(*
  Managing a production on a DigiRound machine.
*)
FUNCTION_BLOCK FB_ProdManager_DMAX EXTENDS FB_BasePrint IMPLEMENTS I_PrintStatusClient, I_ProdManager
VAR
 //references
  _pPU                : POINTER TO FB_PU;               (*PU reference*)
  _pAdsPU             : POINTER TO ST_ADS_PU;
  
  //settings
  _defaultPrintData   : ST_PRINT_SETTING;               (*default PDI data if no CT present*)
  _isVarData          : BOOL; 

  //status
  bPmActive           : BOOL;                           (*a production is active*)
  rfTrig_PmActive     : RF_TRIG;
  lastCreatedCT       : I_CT;                           (*last created container*)

  (*lists*)
  (*--list implementations*)
  prodList            : FB_ListPointerDyn;              (*list fb [pointer to I_CT] - current production elements*)
  _prodMem            : ARRAY[1..lNUM_LIST_SIZE] OF PVOID;   (*list memory for prodList*)
  (*--job trace list*)
  _currJobId          : STRING;                         (*id of current started job*)

  (*internals*)
  _pEcSrc : POINTER TO T_ErrSrc;                                    (*error source definition*)

END_VAR
VAR CONSTANT
  lNUM_LIST_SIZE        : DINT := iCPr_MAX_CONTAINER;   (*number of max. list elements*)
  // other logs
  aC_Dbg_NotReject      : STRING := 'could not rejectNext CT';
  aC_Dbg_InvPtrCT       : STRING := 'invalid pO_ContainerHead';
  aC_Dbg_InvPtrJob      : STRING := 'invalid Job pointer';
  aC_Ddb_GetNext        : STRING := 'getNext from: ';  
END_VAR

IF NOT bInitialized THEN RETURN; END_IF  // ignore

rfTrig_PmActive(CLK:=bPmActive);

(*
  Job was stopped. 
  :return: TRUE if some elements were aborted in machine.
*)
METHOD PRIVATE abortJob : BOOL
VAR
END_VAR
// a job stopped.

// NOTE: not implemented
END_METHOD

PROPERTY bReady : BOOL
GET
bReady := bPmActive;
END_GET
END_PROPERTY

PROPERTY bStarted : BOOL
GET
bStarted := rfTrig_PmActive.RT;
END_GET
END_PROPERTY

PROPERTY bStopped : BOOL
GET
bStopped := rfTrig_PmActive.FT;
END_GET
END_PROPERTY

(*
Create/Build a new container (CT) with next page to be printed.
*)
METHOD CT_Create : BOOL
VAR_INPUT
  sCT            : I_CT;                  // container to produce
END_VAR
VAR 
  _created       : BOOL := FALSE;
  sPage          : ST_PrintPageDef;
END_VAR
// prepare & checks
lastCreatedCT := 0;                      // invalidate last created
IF NOT bInitialized THEN RETURN; END_IF
IF sCT = 0 THEN LogError(aC_Dbg_InvPtrCT); RETURN; END_IF

(* getNext CT *)
IF getNext(sCT := sCT) THEN
  
  // define printer output
  sPage := sCT.sPageDef;
  IF    sPage.lType = EN_PrintPageType.maintenance THEN // - maintenance
    sCT.pCT^.lPrOutput := EN_PrinterOutput.trash;     // -> eject trash
  ELSIF sPage.lType = EN_PrintPageType.production OR   // - production
        sPage.lSrc = EN_PrintPageSrc.overprod OR       // - over-production
        sPage.lType = EN_PrintPageType.separator THEN  // - separator 
    sCT.pCT^.lPrOutput := EN_PrinterOutput.prod;      // -> production output
  ELSE                                                // - rest
    sCT.pCT^.lPrOutput := EN_PrinterOutput.trash;     // -> eject trash
  END_IF

  lastCreatedCT := sCT;                // successfully produced a CT, store last created CT (necessary for async access within this cycle)
  sCT.pCT^.bCreated := TRUE;
  _created := TRUE;
ELSE
  sCT.setError(EC_Print.ecPMInvGetNext, Src:=_pEcSrc^);   // getNext error
END_IF

(* logging *)
LogLvl(Lvl:=E_LogSeverity.Debug, Msg:=CONCAT('create CT: ', sCT.print(0)));

(*return value*)
CT_Create := _created;
END_METHOD

METHOD CT_Finish : BOOL
VAR_INPUT
  sCT            : I_CT;               // container to produce
  bSuccess       : BOOL;               // printed OK?
END_VAR
VAR
  bErr           : BOOL;
END_VAR
(* checks *)
IF NOT bInitialized THEN RETURN; END_IF                             // exit if no production is active
IF sCT = 0 THEN LogError(aC_Dbg_InvPtrCT); RETURN; END_IF  // log invalid pointer 

// remove from production list
IF NOT prodList.RemoveIndex(prodList.FindIndex(sCT.instance)) THEN
  LogError('CT_Finish: could not find CT in prodList'); 
END_IF

// tag machine errors on CT
IF sCT.pCT^.bValid AND NOT bSuccess THEN  
    sCT.setError(EC_Print.ecPMCTMachineErr, Src:=_pEcSrc^);            // tag CT with: error from machine 
END_IF

// report page done to PU
IF NOT sCT.pCT^.bReported AND sCT.pJob <> 0 THEN
  IF _pPU^.endPage(sCT:=sCT, bSuccess:=bSuccess) THEN
    ;
  ELSE
    sCT.setError(EC_Print.ecPMInvSet, Src:=_pEcSrc^);
  END_IF
END_IF

(* logging *)
IF bSuccess THEN
  LogLvl(Lvl:=E_LogSeverity.Detail, Msg:=CONCAT('successCT: ', sCT.print(0)));
ELSE
  LogLvl(Lvl:=E_LogSeverity.Detail, Msg:=CONCAT('eject  CT: ', sCT.print(0)));  
END_IF

(* return value *)
CT_Finish := TRUE;
END_METHOD

(*
  Finalize/Produce a CT. Now we shouldhave all necessary information for configuring the CT.
*)
METHOD CT_Produce : BOOL
VAR_INPUT
  sCT                 : I_CT;               // container to produce
END_VAR
VAR
  _produced           : BOOL := FALSE;
  sPage               : ST_PrintPageDef;
  bPresent            : BOOL;
END_VAR
(* parameter checks *)
IF NOT bInitialized THEN RETURN; END_IF
IF sCT = 0 THEN LogError(aC_Dbg_InvPtrCT); RETURN; END_IF

sCT.pCT^.bValid           := TRUE;                (* we have all data - CT is valid configured*)

// reject page if no container present or overproduction
sPage := sCT.sPageDef;
bPresent := sCT.pCT^.bProductPresent;
IF NOT bPresent AND sPage.lSrc <> EN_PrintPageSrc.overprod  THEN
  (*   add it to rejected queue (high prio reproduction), we will try to produce this CT in next cycle*)
  IF NOT _pPU^.rejPage(sCT:=sCT) THEN
    LogLvl(Lvl:=E_LogSeverity.Info, aC_Dbg_NotReject);
  END_IF
END_IF

(* logging *)
IF bPresent THEN LogLvl(Lvl:=E_LogSeverity.Detail,  Msg:=CONCAT('produceCT: ', sCT.print(0)));
            ELSE LogLvl(Lvl:=E_LogSeverity.Debug,   Msg:=CONCAT('produceCT: ', sCT.print(0))); END_IF

(* return value*)
CT_Produce := _produced;
END_METHOD

PROPERTY defaultPrData : ST_PRINT_SETTING
GET
defaultPrData := _defaultPrintData;
END_GET
END_PROPERTY

METHOD PRIVATE dynAddPage : BOOL
VAR_INPUT
  lType     : EN_PrintPageType; 
  lPageNr   : UDINT;
END_VAR
IF _pPU = 0 THEN F_Report_Error(ErrType:=EN_REPORT_ERROR_TYPE.Report_Error_0Pointer); RETURN; END_IF
IF lType <> EN_PrintPageType.maintenance THEN
  LogError('dynAddPage: only supports maintenance pages'); 
END_IF

_pPU^.addPage(lMaintPageNr:=lPageNr);
END_METHOD

(*
  get next page to be printed.
  :return:    TRUE if success.
*)
METHOD PRIVATE getNext : BOOL               (*get next image to be printed*)
VAR_INPUT
  sCT               : I_CT;                 (*container handle*)
END_VAR
VAR
  bErr              : BOOL;
  lRemainingPages   : UDINT;
END_VAR
VAR_INST
  rTrig_PreStop     : R_TRIG;
END_VAR
IF NOT bInitialized THEN RETURN; END_IF                    (* Exit if no production is active*)

// ask pu for a next page
bErr := NOT _pPU^.getPage(sCT:=sCT, lPagesLeft=>lRemainingPages);

// add to producing list
IF NOT prodList.AddItem(Item := sCT.instance) THEN 
  LogError('getNext: could not add CT to prodList');
  bErr := TRUE;
END_IF

getNext := NOT bErr;
END_METHOD

METHOD init : BOOL
VAR_INPUT
  pPU     : POINTER TO FB_PU;
  pAdsPU  : POINTER TO ST_ADS_PU;
  // machine specific
END_VAR
// parameter checks
IF pPU = 0 OR pAdsPU = 0 THEN
  F_Report_Error(ErrType:=EN_REPORT_ERROR_TYPE.Report_Error_0Pointer);
  RETURN;
END_IF

// register external references
_pPU := pPU;
_pAdsPU := pAdsPU;

// init lists
prodList(List:=_prodMem);  // initial call for list setup and init
prodList.Clear();

// init error source
_pEcSrc := ErrorCodes.fbErrCodeMngr.registerErrSource(
  nLocId:=0, 
  aInstPath:=InstanceName, 
  aLocDescr:='PrintManager DMAX'
);
IF _pEcSrc = 0 THEN LogError('could not register error source'); END_IF

//reset setates
bPmActive := FALSE;
lastCreatedCT := 0;

bInitialized := TRUE;
END_METHOD

METHOD JobFinished : BOOL
VAR_INPUT
  aSeparatorId   : STRING;
END_VAR
// Job Handling -----------------------

// NOTE: nothing implemented for now
END_METHOD

PROPERTY lastCreated : I_CT
GET
lastCreated := lastCreatedCT;
END_GET
END_PROPERTY

METHOD mJobPause
END_METHOD

METHOD mJobStart
VAR_INPUT
	sJobDef	: I_JobDefinition;
END_VAR
IF NOT bInitialized THEN RETURN; END_IF
IF sJobDef = 0 THEN RETURN; END_IF

// start job 
LogLvl(lvl:=E_LogSeverity.Detail, Msg:=F_Concat5('PM start job: ', sJobDef.aJobId, ' (', sJobDef.aJobName, ')'));

// setup PrintManager with new job
_currJobId := sJobDef.aJobId;
_isVarData := sJobDef.isVarData();

// -- init last created
lastCreatedCT := 0;

// -- init defaultPrintData (TODO: not sure why we really need this)
MEMSET(ADR(_defaultPrintData), 0, SIZEOF(_defaultPrintData));   // reset default data

// -- add pre-production pages (product specific) -> maintenance pages
(*FOR lCt := 1 TO lStartEject DO 
  dynAddPage(lType:=EN_PrintPageType.maintenance, 1);
END_FOR*)

bPmActive := TRUE;
END_METHOD

METHOD mJobStop
VAR_INPUT
	sStatus	: I_JobStatus;
END_VAR
VAR
  eHandlingState  : EN_JobHandlingState;
END_VAR
IF NOT bInitialized THEN RETURN; END_IF

(*Stop job*)
LogLvl(lvl:=E_LogSeverity.Detail, Msg:=
  F_Concat7(
    'PM stop job P(',
    TO_STRING(sStatus.iJobProgress.lProductionCount), ') M(',
    TO_STRING(sStatus.iJobProgress.lMaintenanceCount), ') S(',
    TO_STRING(sStatus.iJobProgress.lScrapCount), ')'
  )
);

abortJob();

bPmActive := FALSE;
lastCreatedCT := 0;
END_METHOD

METHOD mProduced
VAR_INPUT
	(* current progress*)
	sProgress	: I_JobProgress;
END_VAR
IF NOT bInitialized THEN RETURN; END_IF
END_METHOD

END_FUNCTION_BLOCK

(* stored: Version 1.1.0.1, ProductVersion 3.1.4024.11
   POU FB_ProdManager_DMAX: Id {6b328657-811b-4dd9-b1f4-d06c9d97af12}, SpecialFunc None
   Folder I_PrintStatusClient: Id {01602ff5-4961-4770-a9e0-df788cccf137}
   Folder I_ProdManager: Id {098fb917-a473-45be-aa26-2a7289011cb1}
   Method abortJob: Id {0b86ce5b-6645-4e9f-88e0-e4df53c97f50}
   Property bReady: Id {33904276-4cf8-4fbb-8168-623dee2f352a}
   Get Get: Id {af74f0be-4916-4823-851b-eec52ffc9c35}
   Property bStarted: Id {003fc039-2ae1-47e7-939b-8b964c2b0215}
   Get Get: Id {77fefb97-cf9a-4c80-ad83-797fc7c7e415}
   Property bStopped: Id {c4f65a10-a22d-442c-b452-0ef8920e8a23}
   Get Get: Id {4ab745ce-3e15-428d-bfcf-e8babe4e4e7a}
   Method CT_Create: Id {db8229d9-012f-45ec-9895-5d9df89c144e}
   Method CT_Finish: Id {7fbbcc1d-cc92-478b-8cc6-a0a3756f5d60}
   Method CT_Produce: Id {9e3a46dc-7f8e-4f60-8028-450ec410f1c3}
   Property defaultPrData: Id {0f30a3d3-bbde-49dd-b640-35e97b7021cb}
   Get Get: Id {6d19f315-df2f-4d12-8181-34118b946600}
   Method dynAddPage: Id {4e3f409c-045d-46ae-bef1-54a6c3ec3f52}
   Method getNext: Id {5d75c39d-9fb1-4ff9-a5b0-edf19030c563}
   Method init: Id {d77ef565-b96f-4032-8974-a22386a23d45}
   Method JobFinished: Id {f266638a-b068-4c56-b67c-8fc6bd6c2d2b}
   Property lastCreated: Id {0d8dadff-1b2d-4f94-a1be-d8278fcd8c5e}
   Get Get: Id {3da8089e-1cda-4562-8078-aa66d5961270}
   Method mJobPause: Id {6a44bd3a-ab99-45aa-ab8c-fcd698bd816f}
   Method mJobStart: Id {c9bb6b9d-7a22-4528-839b-20c5010c2a55}
   Method mJobStop: Id {21a0faba-df46-4fc9-95e9-89fdc44492f2}
   Method mProduced: Id {db99b749-d6ca-4154-97fa-adccf70dbc59} *)
